PROGRAM MAIN
VAR
	
END_VAR

GVL.DataToHmi.LifeBit			:= GVL.DataFromHmi.LifeBit;
GVL.DataToHmi.TestArray			:= GVL.DataFromHmi.TestArray;
GVL.DataToHmi.TestDouble		:= GVL.DataFromHmi.TestDouble;
GVL.DataToHmi.TestString		:= GVL.DataFromHmi.TestString;

END_PROGRAM

(* stored: Version 1.1.0.1, ProductVersion 3.1.4024.16
   POU MAIN: Id {abc9f6d7-23f5-498e-b48b-d5e9ec6e522b}, SpecialFunc None *)
